Staubli VAL3: setVel.pgx

program setVel(num x_nVelType, frame x_fVelFrm, tool x_tTool, mdesc x_mMdesc, num& x_nCmd[])
  local num l_ni
begin
  //choose the type
  switch x_nVelType
    case 1
      $velTool(x_tTool,x_mMdesc)
    break
    case 2
      $velJoint(x_tTool,x_mMdesc)
    break
    default
      $velFrame(x_fVelFrm,x_tTool,x_mMdesc)
    break
  endSwitch
  //
  while true
    $setVelCmd(x_nCmd)
    delay(0)
  endWhile
end
